PROGRAM pouMsgS5
VAR
	
	
	
END_VAR

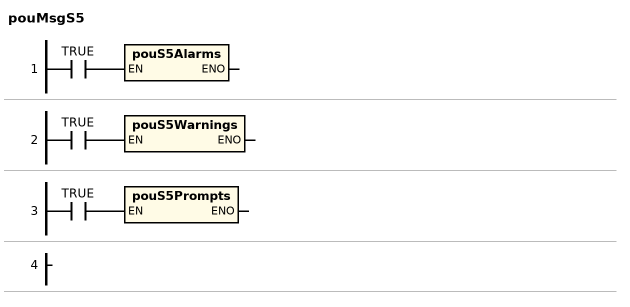
// NETWORK 1
pouS5Alarms();

// NETWORK 2
pouS5Warnings();

// NETWORK 3
pouS5Prompts();

// NETWORK 4

END_PROGRAM

(* stored: Version 1.1.0.1, ProductVersion 3.1.4024.12
   POU pouMsgS5: Id {687acc17-4408-47f9-bc17-4245741e120b}, SpecialFunc None *)
